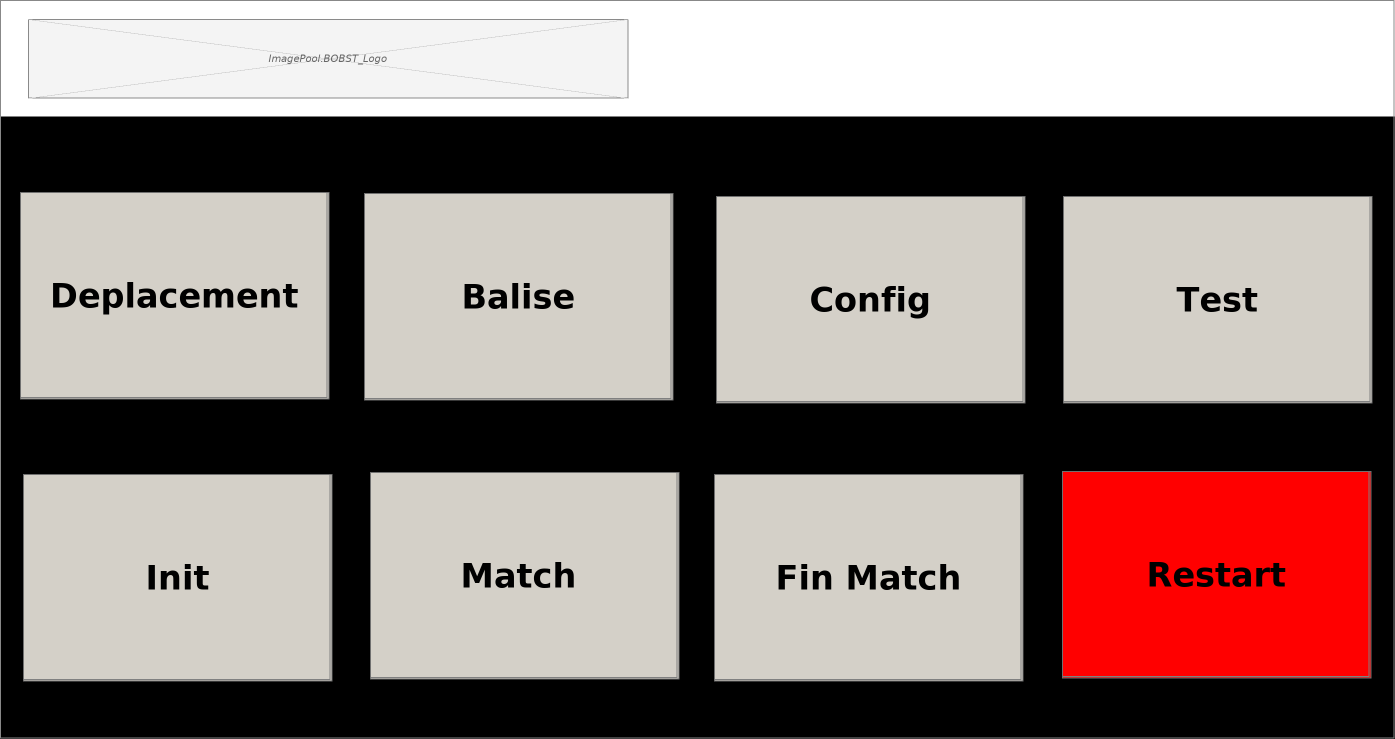
VISUALIZATION V_Menu  // 1395x739
    Rectangle (0,0 1396x116)
    Button (20,192 309x207), "Deplacement"
        OnMouseClick: change screen: V_Deplacement
    Image (28,19 600x79), image: ImagePool.BOBST_Logo
    Button (364,193 309x207), "Balise"
        OnMouseClick: change screen: V_Balise
    Button (716,196 309x207), "Config"
        OnMouseClick: change screen: V_Config
    Button (370,472 309x207), "Match"
        OnMouseClick: change screen: V_Match
    Button (23,474 309x207), "Init"
        OnMouseClick: change screen: V_Init
    Button (714,474 309x207), "Fin Match"
        OnMouseClick: change screen: V_Fin_Match
    Button (1063,196 309x207), "Test"
        OnMouseClick: change screen: V_Test
    Button (1062,471 309x207), "Restart"
        OnMouseClick: toggle G_Visus.bMenuRestart
END_VISUALIZATION

(* stored: Version 1.1.0.1, ProductVersion 3.1.4024.11
   Visu V_Menu: Id {c1f5c3b1-4899-4e18-8f01-2e65675d269e} *)
